TYPE ST_TO_HMI :
STRUCT
	Data		: ST_DATA;
END_STRUCT
END_TYPE

(* stored: Version 1.1.0.1, ProductVersion 3.1.4022.11
   DUT ST_TO_HMI: Id {9757e010-39f6-447d-9bfc-f33a5b91da09} *)
